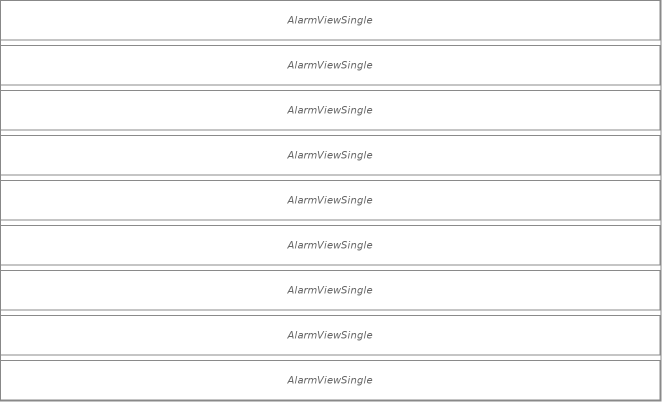
VISUALIZATION AlarmViewMulti  // 662x402
VAR_IN_OUT
	alarm_view: AlarmViewLogger;
END_VAR
    Frame (0,0 660x40), input disabled if: alarm_view.events[1].level = EventLevel.NONE
        shows AlarmViewSingle(event_message := alarm_view.events[1])
    Frame (0,45 660x40), input disabled if: alarm_view.events[2].level = EventLevel.NONE
        shows AlarmViewSingle(event_message := alarm_view.events[2])
    Frame (0,90 660x40), input disabled if: alarm_view.events[3].level = EventLevel.NONE
        shows AlarmViewSingle(event_message := alarm_view.events[3])
    Frame (0,135 660x40), input disabled if: alarm_view.events[4].level = EventLevel.NONE
        shows AlarmViewSingle(event_message := alarm_view.events[4])
    Frame (0,180 660x40), input disabled if: alarm_view.events[5].level = EventLevel.NONE
        shows AlarmViewSingle(event_message := alarm_view.events[5])
    Frame (0,225 660x40), input disabled if: alarm_view.events[6].level = EventLevel.NONE
        shows AlarmViewSingle(event_message := alarm_view.events[6])
    Frame (0,270 660x40), input disabled if: alarm_view.events[7].level = EventLevel.NONE
        shows AlarmViewSingle(event_message := alarm_view.events[7])
    Frame (0,315 660x40), input disabled if: alarm_view.events[8].level = EventLevel.NONE
        shows AlarmViewSingle(event_message := alarm_view.events[8])
    Frame (0,360 660x40), input disabled if: alarm_view.events[9].level = EventLevel.NONE
        shows AlarmViewSingle(event_message := alarm_view.events[9])
END_VISUALIZATION

(* stored: Version 1.1.0.1, ProductVersion 3.1.4022.18
   Visu AlarmViewMulti: Id {d5e60cda-2b5b-4af6-902a-b153f8536757} *)
